INTERFACE I_PersistantDataStorage

END_INTERFACE

(* stored: Version 1.1.0.1
   Itf I_PersistantDataStorage: Id {ef419ae2-fd84-4184-8b85-555366ae9e1e} *)
